TYPE ST_Device :
STRUCT
	value : DINT;;
END_STRUCT
END_TYPE

(* stored: Version 1.1.0.1, ProductVersion 3.1.4024.12
   DUT ST_Device: Id {ba879b4d-277a-4798-9204-86999f674d44} *)
